FUNCTION_BLOCK MotVsFailures_HMI (* Service Interface Function Block Type *)
  (* Standard: 61499-2 *)
  (* Version 0.0, 8/5/2026, Schneider Electric, template *)
  PACKAGE SE.Nereda;
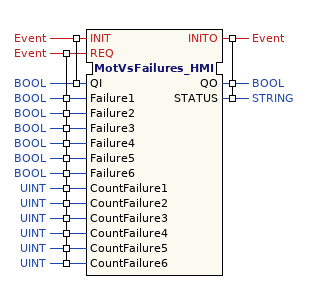
  EVENT_INPUT
    INIT WITH QI;
    REQ WITH Failure1, Failure2, Failure3, Failure4, Failure5, Failure6, CountFailure1, CountFailure2, CountFailure3, CountFailure4, CountFailure5, CountFailure6;
  END_EVENT
  EVENT_OUTPUT
    INITO WITH QO, STATUS;
  END_EVENT
  VAR_INPUT
    QI : BOOL;
    Failure1 : BOOL;
    Failure2 : BOOL;
    Failure3 : BOOL;
    Failure4 : BOOL;
    Failure5 : BOOL;
    Failure6 : BOOL;
    CountFailure1 : UINT;
    CountFailure2 : UINT;
    CountFailure3 : UINT;
    CountFailure4 : UINT;
    CountFailure5 : UINT;
    CountFailure6 : UINT;
  END_VAR
  VAR_OUTPUT
    QO : BOOL; (* Event Output Qualifier *)
    STATUS : STRING; (* Service Status *)
  END_VAR
  SERVICE /
    SEQUENCE 
    END_SEQUENCE
  END_SERVICE
END_FUNCTION_BLOCK
